// this class is following the OOP Desgn Pattern of a builder (max str length 255)
FUNCTION_BLOCK WSJSONStringBuilder_t
VAR_INPUT
END_VAR
VAR_OUTPUT
END_VAR
VAR
	_str : STRING(2000) := '';
END_VAR

METHOD addAttributeBool : BOOL
VAR_INPUT
	key : STRING(255);
	value : BOOL;
END_VAR
addAttributeBool := addAttributeString(key, BOOL_TO_STRING(value));
return;
END_METHOD

METHOD addAttributeINT : BOOL
VAR_INPUT
	key: STRING(255);
	value: INT;
END_VAR
VAR
	_keyValuePair: STRING(255);
	_tmpStr: STRING(255);
END_VAR
_keyValuePair := formateAttributeINT(key, value);

IF  _keyValuePair = 'ERROR' OR len(_str) + len(_keyValuePair) + 2 > 2000 THEN // length of existing string + new keyValuePar + '{' + '}'
	addAttributeINT := FALSE; 
	RETURN;
END_IF

_tmpStr := concat(_keyValuePair, ',');
concat2(ADR(_str), ADR(_tmpStr), ADR(_str), 2000); // apped key value pair to string with ',' at the end
//_str := concat(_str, concat(_keyValuePair, ',')); // apped key value pair to string with ',' at the end

addAttributeINT := TRUE;
RETURN;
END_METHOD

// adds an attribute (if it returns true: succsess, if false: failed)
METHOD addAttributeString : BOOL
VAR_INPUT
	key : STRING(255);
	value : STRING(255);
END_VAR
VAR
	_tmpStr : STRING := '';
	_keyValuePair : STRING := '';
END_VAR
_keyValuePair := formateAttribute(key, value);

IF  _keyValuePair = 'ERROR' OR len(_str) + len(_keyValuePair) + 2 > 2000 THEN // length of existing string + new keyValuePar + '{' + '}'
	addAttributeString := FALSE; 
	RETURN;
END_IF

_tmpStr := concat(_keyValuePair, ',');
concat2(ADR(_str), ADR(_tmpStr), ADR(_str), 2000); // apped key value pair to string with ',' at the end
//_str := concat(_str, concat(_keyValuePair, ',')); 

addAttributeString := TRUE;
RETURN;
END_METHOD

// builds the JSON string (if it fails output = 'ERROR')
METHOD build : STRING(1000)
VAR_INPUT
END_VAR
VAR
	_lastCharOfStr : STRING(1) := '';
	_appendStr : STRING(1) := '}';
	_prefixStr : STRING(1) := '{';
END_VAR
IF len(_str) + 1 > 2000 OR _str = '' THEN // validate data
	build := 'ERROR';
	RETURN;
END_IF

//_lastCharOfStr := right(_str, 1);

//IF _lastCharOfStr = ',' THEN // check if last character is a ','
delete2(ADR(_str), ADR(_str), 2000, 1, len2(ADR(_str)));
	//_str := delete(_str, 1, len(_str));
//END_IF

// wrap key value pair list

CONCAT2(ADR(_prefixStr), ADR(_str), ADR(_str), 2000); 
CONCAT2(ADR(_str), ADR(_appendStr), ADR(build), 2000); 
//build := concat('{', concat(_str, '}'));
RETURN;
END_METHOD

// clears whole attribute buffer
METHOD clear : BOOL
VAR_INPUT
END_VAR
_str := '';
END_METHOD

// takes a key and attribute and formats it to a valid key value pair (if string is too long ouput will be 'ERROR')
METHOD PRIVATE formateAttribute : string(255)
VAR_INPUT
	key : STRING(255);
	value : STRING(255);
END_VAR
VAR
	_tmpStr : STRING(255) := '';
END_VAR
IF LEN(key) + len(value) + 5 > 2000  THEN // return error if string is too long
	formateAttribute := 'ERROR';
	RETURN;
END_IF

// formate key value pair
_tmpStr := concat('"', key);
_tmpStr := concat(_tmpStr, '":"');
_tmpStr := concat(_tmpStr, value);
formateAttribute := concat(_tmpStr, '"');
RETURN;
END_METHOD

METHOD PRIVATE formateAttributeINT : string(255)
VAR_INPUT
	key: STRING(255);
	value: INT;
END_VAR

VAR
	_tmpStr: STRING(255);
END_VAR
IF LEN(key) + len(INT_TO_STRING(value)) + 3 > 2000  THEN // return error if string is too long
	formateAttributeINT := 'ERROR';
	RETURN;
END_IF

// formate key value pair
_tmpStr := concat('"', key);
_tmpStr := concat(_tmpStr, '":');
formateAttributeINT := concat(_tmpStr, INT_TO_STRING(value));
RETURN;
END_METHOD

END_FUNCTION_BLOCK

(* stored: Version 1.1.0.1
   POU WSJSONStringBuilder_t: Id {d98c2455-b240-4706-869a-ec781ba7607c}, SpecialFunc None
   Method addAttributeBool: Id {1cae107d-e885-4445-98b1-3989eb7af2ae}
   Method addAttributeINT: Id {87243de8-59af-422c-b4fc-4c8733f2c3c1}
   Method addAttributeString: Id {c7fed67b-ada5-4e34-9fc1-b0c345e3d063}
   Method build: Id {94f97329-dfda-4a70-8dfb-7a8101409cc9}
   Method clear: Id {8260fd64-4ef9-4618-b489-3c2279a8acf5}
   Method formateAttribute: Id {3d3b34e3-3e57-42ba-9ccb-2b9217efffe2}
   Method formateAttributeINT: Id {724a82b9-7e58-420a-8d4e-582703e6e720} *)
